// TIA Portal project "Pressure control in a reciever" (V16)

(* hardware
DEVICE "S7-1200 station_2"  S7-1200 Station
   slot 0: "Rack_0"  S7-1200 Rack  Rack  V1.0
   slot 1: "PLC_2"  CPU 1212C DC/DC/DC  6ES7 212-1AE40-0XB0  V4.4
*)

// ===== PLC "PLC_2"  CPU 1212C DC/DC/DC =====

VAR_GLOBAL   // PLC tag table "Default tag table"
   "90 PSI Switch bit" AT %M0.0 : Bool;
   "110 PSI Switch bit" AT %M0.1 : Bool;
   "Pump Energize bit" AT %M0.2 : Bool;
   "Run Indicator Light energize bit" AT %M0.3 : Bool;
   "pump trigger" AT %M0.4 : Bool;
   "Indicator light trigger" AT %M0.5 : Bool;
   "90 PSI Switch" AT %I0.0 : Bool;
   "110 PSI Switch" AT %I0.1 : Bool;
   "Pump Output" AT %Q0.0 : Bool;
   "Run Indicator Light" AT %Q0.1 : Bool;
   "Pressure Level" AT %MW2 : Int;
   "ONS1" AT %M1.2 : Bool;
   "ONS2" AT %M1.3 : Bool;
   "Pump Interrupt" AT %M0.6 : Bool;
   "Light Interrupt" AT %M0.7 : Bool;
END_VAR

DATA_BLOCK "Control logic_DB"   // DB1
{ S7_Optimized_Access := 'TRUE' }
VERSION : 0.1
// stored: InstanceOfName Control logic LAD
"Control logic LAD"
BEGIN
END_DATA_BLOCK

DATA_BLOCK "IO_DB_1"   // DB3
{ S7_Optimized_Access := 'TRUE' }
VERSION : 0.1
// stored: InstanceOfName IO LAD
"IO LAD"
BEGIN
END_DATA_BLOCK

DATA_BLOCK "Pump Cycle_DB"   // DB5
{ S7_Optimized_Access := 'TRUE' }
VERSION : 0.1
// stored: InstanceOfName Pump Cycle LAD
"Pump Cycle LAD"
BEGIN
END_DATA_BLOCK

// folder: System blocks/Program resources

DATA_BLOCK "IEC_Timer_0_DB"   // DB2
{ S7_Optimized_Access := 'TRUE' }
AUTHOR : Simatic
FAMILY : IEC
NAME : IEC_TMR
VERSION : 1.0
// stored: InstanceOfName IEC_TIMER
"IEC_TIMER"
BEGIN
END_DATA_BLOCK

DATA_BLOCK "IEC_Timer_0_DB_1"   // DB4
{ S7_Optimized_Access := 'TRUE' }
AUTHOR : Simatic
FAMILY : IEC
NAME : IEC_TMR
VERSION : 1.0
// stored: InstanceOfName IEC_TIMER
"IEC_TIMER"
BEGIN
END_DATA_BLOCK

DATA_BLOCK "IEC_Timer_0_DB_2"   // DB6
{ S7_Optimized_Access := 'TRUE' }
AUTHOR : Simatic
FAMILY : IEC
NAME : IEC_TMR
VERSION : 1.0
// stored: InstanceOfName IEC_TIMER
"IEC_TIMER"
BEGIN
END_DATA_BLOCK

DATA_BLOCK "IEC_Timer_0_DB_3"   // DB7
{ S7_Optimized_Access := 'TRUE' }
AUTHOR : Simatic
FAMILY : IEC
NAME : IEC_TMR
VERSION : 1.0
// stored: InstanceOfName IEC_TIMER
"IEC_TIMER"
BEGIN
END_DATA_BLOCK

DATA_BLOCK "IEC_Timer_0_DB_4"   // DB8
{ S7_Optimized_Access := 'TRUE' }
AUTHOR : Simatic
FAMILY : IEC
NAME : IEC_TMR
VERSION : 1.0
// stored: InstanceOfName IEC_TIMER
"IEC_TIMER"
BEGIN
END_DATA_BLOCK

DATA_BLOCK "IEC_Timer_0_DB_5"   // DB9
{ S7_Optimized_Access := 'TRUE' }
AUTHOR : Simatic
FAMILY : IEC
NAME : IEC_TMR
VERSION : 1.0
// stored: InstanceOfName IEC_TIMER
"IEC_TIMER"
BEGIN
END_DATA_BLOCK

DATA_BLOCK "IEC_Timer_0_DB_6"   // DB10
{ S7_Optimized_Access := 'TRUE' }
AUTHOR : Simatic
FAMILY : IEC
NAME : IEC_TMR
VERSION : 1.0
// stored: InstanceOfName IEC_TIMER
"IEC_TIMER"
BEGIN
END_DATA_BLOCK

DATA_BLOCK "IEC_Timer_0_DB_7"   // DB11
{ S7_Optimized_Access := 'TRUE' }
AUTHOR : Simatic
FAMILY : IEC
NAME : IEC_TMR
VERSION : 1.0
// stored: InstanceOfName IEC_TIMER
"IEC_TIMER"
BEGIN
END_DATA_BLOCK

// folder: (top level)

FUNCTION_BLOCK "IO LAD"   // FB1, LAD
{ S7_Optimized_Access := 'TRUE' }
VERSION : 0.1
BEGIN

REGION Network 1
   // Inputs
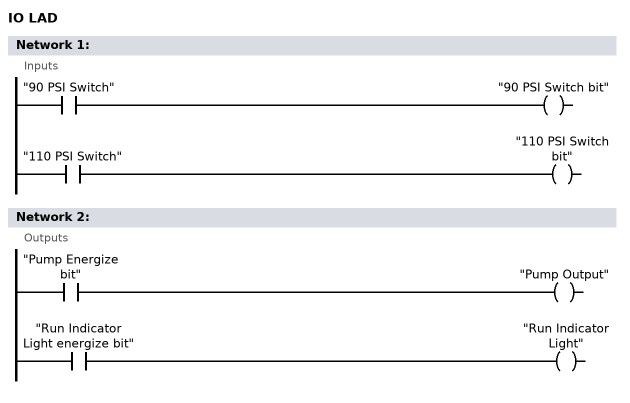
   RUNG wire#powerrail
      Contact( "90 PSI Switch" )
      Coil( "90 PSI Switch bit" )
   END_RUNG
   RUNG wire#powerrail
      Contact( "110 PSI Switch" )
      Coil( "110 PSI Switch bit" )
   END_RUNG
   // the same network as SCL:
   "90 PSI Switch bit" := "90 PSI Switch";
   "110 PSI Switch bit" := "110 PSI Switch";
END_REGION

REGION Network 2
   // Outputs
   RUNG wire#powerrail
      Contact( "Pump Energize bit" )
      Coil( "Pump Output" )
   END_RUNG
   RUNG wire#powerrail
      Contact( "Run Indicator Light energize bit" )
      Coil( "Run Indicator Light" )
   END_RUNG
   // the same network as SCL:
   "Pump Output" := "Pump Energize bit";
   "Run Indicator Light" := "Run Indicator Light energize bit";
END_REGION
END_FUNCTION_BLOCK

FUNCTION_BLOCK "Control logic LAD"   // FB2, LAD
{ S7_Optimized_Access := 'TRUE' }
VERSION : 0.1
// For the control of both the pump and the indicator light, the digital control logic has been implemented in the code for the safety of the devices, since the switches can flicker on/off several times within a very short period of time. This flickering could eventually lead to the failure of the electrical devices.
   VAR
      "ONS 1" : Bool;
   END_VAR
   VAR_TEMP   // added for the SCL form of the ladder/FBD networks
      _w1 : Bool;
   END_VAR
BEGIN

REGION Network 1
   // Pump control logic- The pump will be energized (run) as long as the pressure inside the reciever (container) remains below than 110 PSI
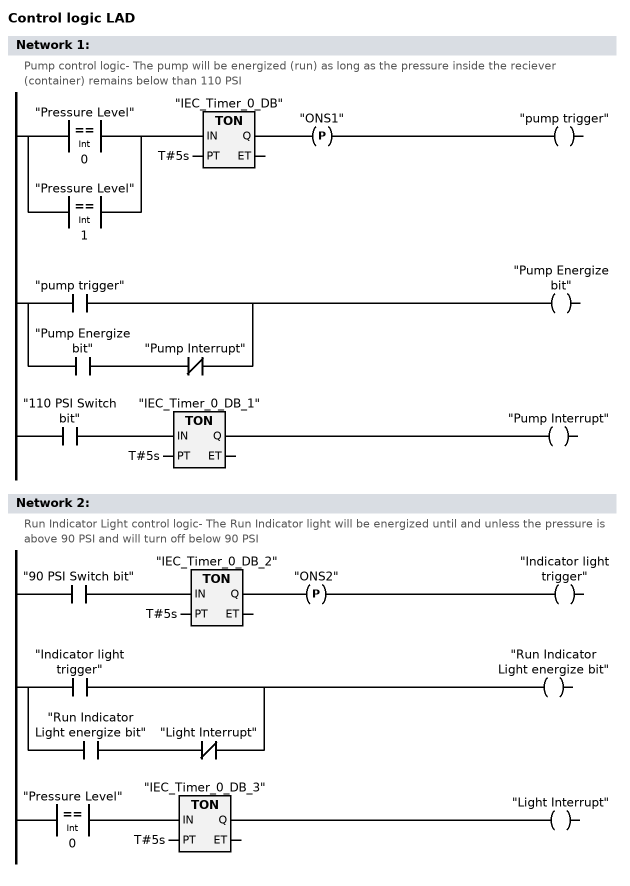
   "IEC_Timer_0_DB".TON(IN := ("Pressure Level" = 0) OR ("Pressure Level" = 1), PT := T#5s);
   #_w1 := "IEC_Timer_0_DB".Q AND NOT "ONS1";   // rising edge
   "ONS1" := "IEC_Timer_0_DB".Q;
   "pump trigger" := #_w1;
   "Pump Energize bit" := "pump trigger" OR ("Pump Energize bit" AND NOT "Pump Interrupt");
   "IEC_Timer_0_DB_1".TON(IN := "110 PSI Switch bit", PT := T#5s);
   "Pump Interrupt" := "IEC_Timer_0_DB_1".Q;
END_REGION

REGION Network 2
   // Run Indicator Light control logic- The Run Indicator light will be energized until and unless the pressure is above 90 PSI and will turn off below 90 PSI
   "IEC_Timer_0_DB_2".TON(IN := "90 PSI Switch bit", PT := T#5s);
   #_w1 := "IEC_Timer_0_DB_2".Q AND NOT "ONS2";   // rising edge
   "ONS2" := "IEC_Timer_0_DB_2".Q;
   "Indicator light trigger" := #_w1;
   "Run Indicator Light energize bit" := "Indicator light trigger" OR ("Run Indicator Light energize bit" AND NOT "Light Interrupt");
   "IEC_Timer_0_DB_3".TON(IN := "Pressure Level" = 0, PT := T#5s);
   "Light Interrupt" := "IEC_Timer_0_DB_3".Q;
END_REGION
END_FUNCTION_BLOCK

FUNCTION_BLOCK "Pump Cycle LAD"   // FB3, LAD
{ S7_Optimized_Access := 'TRUE' }
VERSION : 0.1
// Increase and decrease of pressure in the container takes place in a cycle. Initially, the container has pressure below 90 PSI. Once the pump start increasing the pressure such that it reaches 110 PSI, the pump stops and remains off until the pressure again decreases below 90 PSI.
BEGIN

REGION Network 1
   // Pressure Level:
   // 0 = Pressure below 90 PSI
   // 1 = Pressure between 110 PSI and 90 PSI and container is being pressurized
   // 2 = Pressure above 110 PSI 
   // 3 = Pressure between 110 PSI and  90  PSI and pressure is decreasing in container
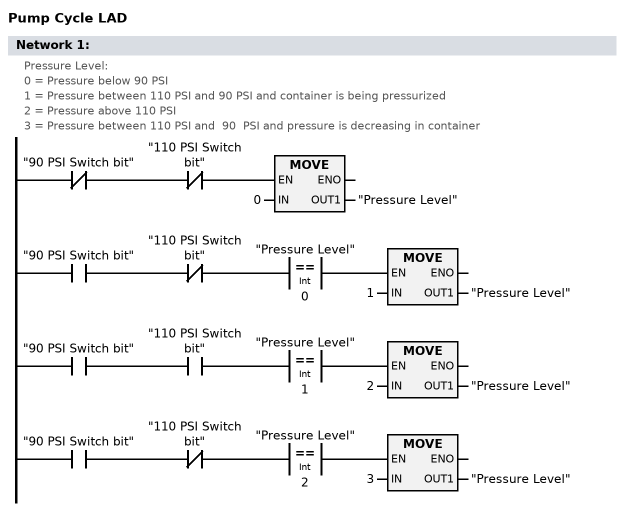
   RUNG wire#powerrail
      I_Contact( "90 PSI Switch bit" )
      I_Contact( "110 PSI Switch bit" )
      Move(in := 0, out1 => "Pressure Level")
   END_RUNG
   RUNG wire#powerrail
      Contact( "90 PSI Switch bit" )
      I_Contact( "110 PSI Switch bit" )
      { S7_Templates := "SrcType := Int" } EQ_Contact(in1 := "Pressure Level", in2 := 0)
      Move(in := 1, out1 => "Pressure Level")
   END_RUNG
   RUNG wire#powerrail
      Contact( "90 PSI Switch bit" )
      Contact( "110 PSI Switch bit" )
      { S7_Templates := "SrcType := Int" } EQ_Contact(in1 := "Pressure Level", in2 := 1)
      Move(in := 2, out1 => "Pressure Level")
   END_RUNG
   RUNG wire#powerrail
      Contact( "90 PSI Switch bit" )
      I_Contact( "110 PSI Switch bit" )
      { S7_Templates := "SrcType := Int" } EQ_Contact(in1 := "Pressure Level", in2 := 2)
      Move(in := 3, out1 => "Pressure Level")
   END_RUNG
   // the same network as SCL:
   IF NOT "90 PSI Switch bit" AND NOT "110 PSI Switch bit" THEN "Pressure Level" := 0; END_IF;
   IF "90 PSI Switch bit" AND NOT "110 PSI Switch bit" AND ("Pressure Level" = 0) THEN
       "Pressure Level" := 1;
   END_IF;
   IF "90 PSI Switch bit" AND "110 PSI Switch bit" AND ("Pressure Level" = 1) THEN
       "Pressure Level" := 2;
   END_IF;
   IF "90 PSI Switch bit" AND NOT "110 PSI Switch bit" AND ("Pressure Level" = 2) THEN
       "Pressure Level" := 3;
   END_IF;
END_REGION
END_FUNCTION_BLOCK

FUNCTION_BLOCK "Control logic FBD"   // FB4, FBD
{ S7_Optimized_Access := 'TRUE' }
VERSION : 0.1
   VAR_TEMP   // added for the SCL form of the ladder/FBD networks
      _w1 : Bool;
   END_VAR
BEGIN

REGION Network 1
   // Pump Control Logic
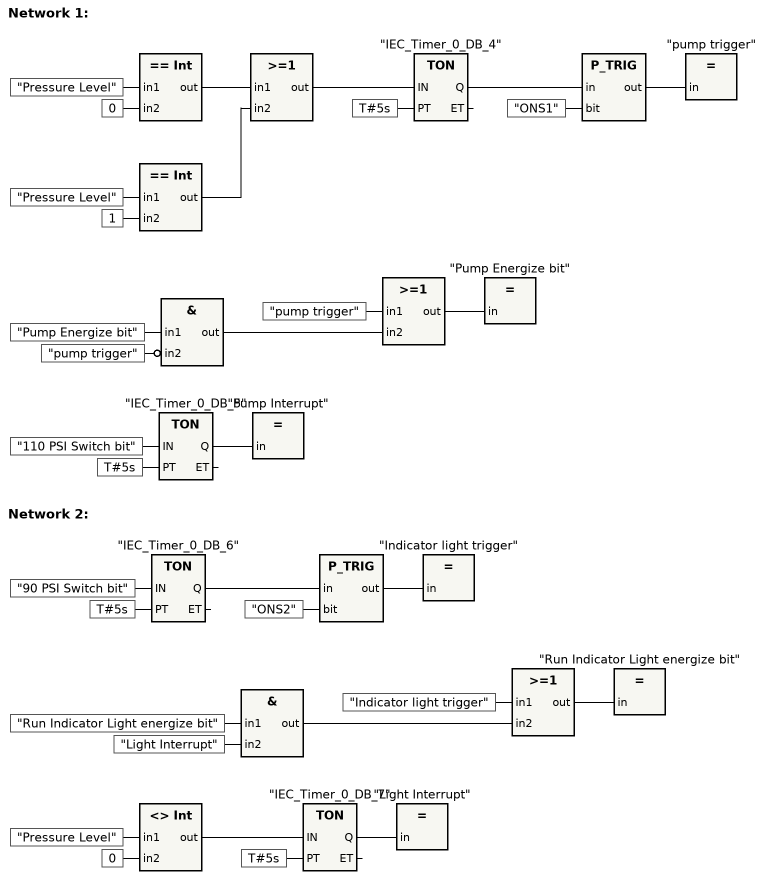
   "IEC_Timer_0_DB_4".TON(IN := ("Pressure Level" = 0) OR ("Pressure Level" = 1), PT := T#5s);
   #_w1 := "IEC_Timer_0_DB_4".Q AND NOT "ONS1";   // rising edge
   "ONS1" := "IEC_Timer_0_DB_4".Q;
   "pump trigger" := #_w1;
   "Pump Energize bit" := "pump trigger" OR ("Pump Energize bit" AND NOT "pump trigger");
   "IEC_Timer_0_DB_5".TON(IN := "110 PSI Switch bit", PT := T#5s);
   "Pump Interrupt" := "IEC_Timer_0_DB_5".Q;
END_REGION

REGION Network 2
   // Run Indicator Light Control Logic
   "IEC_Timer_0_DB_6".TON(IN := "90 PSI Switch bit", PT := T#5s);
   #_w1 := "IEC_Timer_0_DB_6".Q AND NOT "ONS2";   // rising edge
   "ONS2" := "IEC_Timer_0_DB_6".Q;
   "Indicator light trigger" := #_w1;
   "Run Indicator Light energize bit" := "Indicator light trigger" OR ("Run Indicator Light energize bit" AND "Light Interrupt");
   "IEC_Timer_0_DB_7".TON(IN := "Pressure Level" <> 0, PT := T#5s);
   "Light Interrupt" := "IEC_Timer_0_DB_7".Q;
END_REGION
END_FUNCTION_BLOCK

FUNCTION_BLOCK "IO FBD"   // FB5, FBD
{ S7_Optimized_Access := 'TRUE' }
VERSION : 0.1
BEGIN

REGION Network 1
   // Inputs
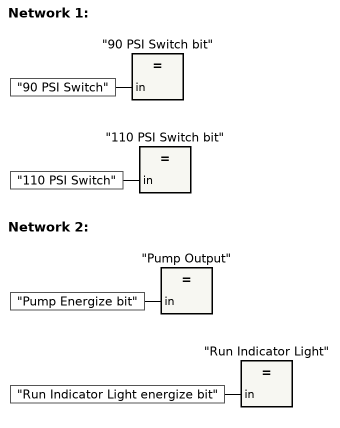
   "90 PSI Switch bit" := "90 PSI Switch";
   "110 PSI Switch bit" := "110 PSI Switch";
END_REGION

REGION Network 2
   // Outputs
   "Pump Output" := "Pump Energize bit";
   "Run Indicator Light" := "Run Indicator Light energize bit";
END_REGION
END_FUNCTION_BLOCK

FUNCTION_BLOCK "Pump Cycle FBD"   // FB6, FBD
{ S7_Optimized_Access := 'TRUE' }
VERSION : 0.1
BEGIN

REGION Network 1
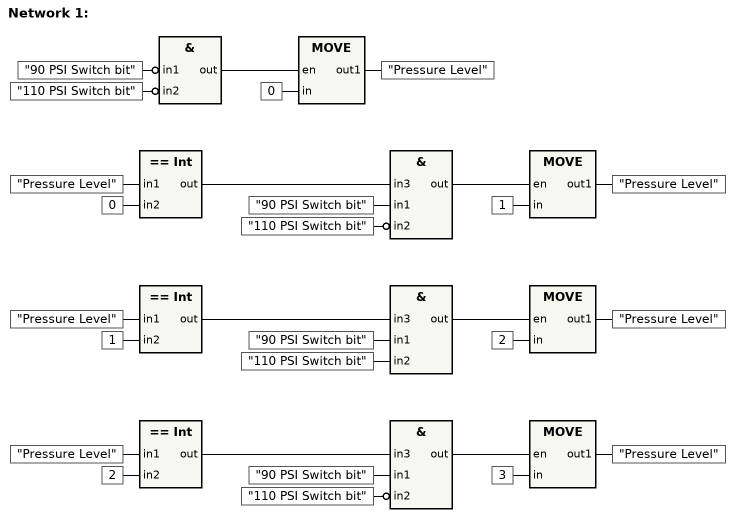
   IF NOT "90 PSI Switch bit" AND NOT "110 PSI Switch bit" THEN "Pressure Level" := 0; END_IF;
   IF ("Pressure Level" = 0) AND "90 PSI Switch bit" AND NOT "110 PSI Switch bit" THEN
       "Pressure Level" := 1;
   END_IF;
   IF ("Pressure Level" = 1) AND "90 PSI Switch bit" AND "110 PSI Switch bit" THEN
       "Pressure Level" := 2;
   END_IF;
   IF ("Pressure Level" = 2) AND "90 PSI Switch bit" AND NOT "110 PSI Switch bit" THEN
       "Pressure Level" := 3;
   END_IF;
END_REGION
END_FUNCTION_BLOCK

ORGANIZATION_BLOCK "Main"   // OB1, LAD, ProgramCycle
TITLE = "Main Program Sweep (Cycle)"
{ S7_Optimized_Access := 'TRUE' }
VERSION : 0.1
// Project explanantion: The project consists of a pump which is used to regulate the pressure in a reciever (container). Inside the container there are two pressure switches (90 PSI switch and 110 PSI). The pump will start if the pressure is below 90 PSI and will turn off once the pressure reaches 110 PSI and remains off until and unless the pressure decreases back to 90 PSI. As soon as the pressure reaches 90 PSI, the Run indicator light turns on and remains on until the pressure decreases below 90 PSI.
// Test Criteria :
// 1) Start simulation, the pump should start immediately but the light should be off.
// 2) Force the 90 PSI switch to 1. The pump should keep on running but the light should turn on.
// 3) Leave the 90 PSI switch to 1 and Force the 110 PSI switch to 1 . The pump should stop running but the light should remain on.
// 4) Leave the 90  PSI switch to 1 and Force the 110 PSI switch to 0. The pump should remain off and the light remains on.
// 5) Force both 90 PSI and 110 PSI switches back to 0. The pump should start back on and the light goes off.
// 
// Note : The code is written both in LAD and FBD
   VAR_INPUT
      Initial_Call : Bool;   // Initial call of this OB
      Remanence : Bool;   // =True, if remanent data are available
   END_VAR
BEGIN

REGION Network 1
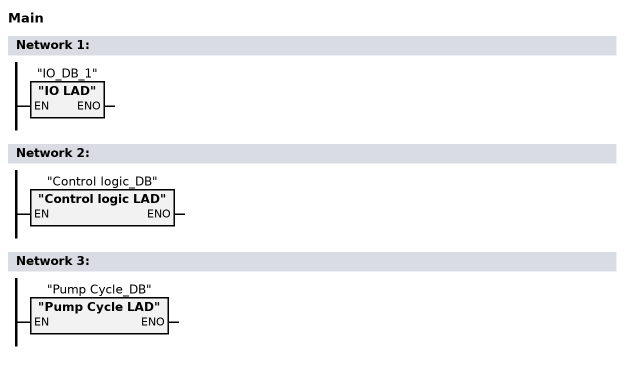
   RUNG wire#powerrail
      "IO_DB_1"()
   END_RUNG
   // the same network as SCL:
   "IO_DB_1"();   // "IO LAD"
END_REGION

REGION Network 2
   RUNG wire#powerrail
      "Control logic_DB"()
   END_RUNG
   // the same network as SCL:
   "Control logic_DB"();   // "Control logic LAD"
END_REGION

REGION Network 3
   RUNG wire#powerrail
      "Pump Cycle_DB"()
   END_RUNG
   // the same network as SCL:
   "Pump Cycle_DB"();   // "Pump Cycle LAD"
END_REGION
END_ORGANIZATION_BLOCK